FUNCTION_BLOCK FB_MAA
VAR_IN_OUT
	fbArbiter: FB_Arbiter;
    fbFFHWO: FB_HardwareFFOutput;
	stYStage: DUT_MotionStage;
	stXStage: DUT_MotionStage;
END_VAR
VAR_INPUT
	 {attribute 'pytmc' := '
        pv: :PMPS:AribterEnabled
        io: io
    '}
	bArbiterEnabled: BOOL:=TRUE;;
	 nTransitionAssertionID: UDINT;
	stAprt1: DUT_PositionState;
	stAprt2: DUT_PositionState;
	stAprt3: DUT_PositionState;
	stAprt4: DUT_PositionState;
	stXCen: DUT_PositionState;
	i_DevName: STRING:= 'AT1K0-MAA';
END_VAR
VAR_OUTPUT	
	 {attribute 'pytmc' := '
        pv: Y:STATE
        io: io
    '}
    fbStates: FB_MAA_States;
	
	{attribute 'pytmc' := '
        pv: X:STATE 
        io: io
    '}
    fbStates_X: FB_MAA_States_X;
END_VAR
VAR

	fbYStage: FB_MotionStage;
	fbXStage: FB_MotionStage;
	
	
	fSize1: REAL:=4; //mm
	fSize2: REAL:=5; //mm
	fSize3: REAL:=7; //mm
	fSize4: REAL:=9; //mm
	
	bInit:BOOL := TRUE;
	tArbiterTimeout: TIME:= T#10S;
	FFO    :    FB_FastFault :=(
        i_DevName := 'AT1K0-MAA',
        i_Desc := 'Fault occurs when the PMPS Aribter is switched off for the aperture plate states BPTM',
        i_TypeCode := 16#1010);
END_VAR

if(bInit) THEN
	stYStage.bHardwareEnable := TRUE;
	stYStage.bPowerSelf := FALSE;
	stYStage.nBrakeMode := ENUM_StageBrakeMode.IF_MOVING;
	stXStage.bHardwareEnable := TRUE;
	stXStage.bPowerSelf := FALSE;
	stXStage.nBrakeMode := ENUM_StageBrakeMode.NO_BRAKE;
	bInit:=FALSE;
	
	// States settings
	stAprt1.nRequestAssertionID := nTransitionAssertionID+1;
	stAprt1.bUseRawCounts := FALSE;
	stAprt1.stBeamParams := PMPS_GVL.cstFullBeam;
	stAprt1.stBeamParams.astApertures[1].Height := fSize1;
	stAprt1.stBeamParams.astApertures[1].Width := fSize1;
	stAprt1.bValid := TRUE;
	
	stAprt2.nRequestAssertionID := nTransitionAssertionID+2;
	stAprt2.bUseRawCounts := FALSE;
	stAprt2.stBeamParams := PMPS_GVL.cstFullBeam;
	stAprt2.stBeamParams.astApertures[1].Height := fSize2;
	stAprt2.stBeamParams.astApertures[1].Width :=fSize2;
	stAprt2.bValid := TRUE;
	
	stAprt3.nRequestAssertionID := nTransitionAssertionID+3;
	stAprt3.bUseRawCounts := FALSE;
	stAprt3.stBeamParams := PMPS_GVL.cstFullBeam;
	stAprt3.stBeamParams.astApertures[1].Height := fSize3;
	stAprt3.stBeamParams.astApertures[1].Width := fSize3;
	stAprt3.bValid := TRUE;
	
	stAprt4.nRequestAssertionID := nTransitionAssertionID+4;
	stAprt4.bUseRawCounts := FALSE;
	stAprt4.stBeamParams := PMPS_GVL.cstFullBeam;
	stAprt4.stBeamParams.astApertures[1].Height := fSize4;
	stAprt4.stBeamParams.astApertures[1].Width := fSize4;
	stAprt4.bValid := TRUE;
	
	stXCen.nRequestAssertionID := nTransitionAssertionID+6;
	stXCen.bUseRawCounts := FALSE;
	stXCen.stBeamParams := PMPS_GVL.cstFullBeam;
	stXCen.bValid := TRUE;
	
	FFO.i_DevName := i_DevName;

END_IF


fbYStage(stMotionStage:=stYStage);
fbXStage(stMotionStage:=stXStage);

fbStates(
	fbArbiter:=fbArbiter,
    fbFFHWO:=fbFFHWO,
    nTransitionAssertionID:=nTransitionAssertionID,
	stTransitionBeam:= PMPS_GVL.cst0RateBeam,
	bArbiterEnabled := bArbiterEnabled,
	tArbiterTimeout :=tArbiterTimeout,
    stMotionStage:=stYStage,
	bEnable:=TRUE,
    stAprt1:=stAprt1,
    stAprt2:=stAprt2,
    stAprt3:=stAprt3,
    stAprt4:=stAprt4);

fbStates_X(
	fbArbiter:=fbArbiter,
    fbFFHWO:=fbFFHWO,
    nTransitionAssertionID:=nTransitionAssertionID+5,
	stTransitionBeam:= PMPS_GVL.cst0RateBeam,
	tArbiterTimeout := tArbiterTimeout,
    stMotionStage:=stXStage,
	bEnable:=TRUE,
    stXCen:=stXCen);


(*FAST FAULT*)
FFO(i_xOK := bArbiterEnabled,
    i_xReset := ,
	i_xAutoReset :=,
    io_fbFFHWO := fbFFHWO);

END_FUNCTION_BLOCK

(* stored: Version 1.1.0.1, ProductVersion 3.1.4022.18
   POU FB_MAA: Id {8c4640db-3bb7-4671-b4ea-e9d46c4b8221}, SpecialFunc None *)
